TYPE ST_PNOZRawOut :
STRUCT
    aByte : ARRAY[1..19] OF BYTE;
END_STRUCT
END_TYPE

(* stored: Version 1.1.0.1
   DUT ST_PNOZRawOut: Id {f721d84d-ba9b-4caa-9515-51e70651d496} *)
